(* PLC project  *)

PROGRAM P

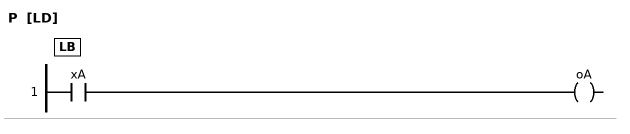
(* LD diagram, written out as Structured Text *)
LA:
(* second one *)
LB:
oA := xA;
END_PROGRAM
